TYPE ST185_Cylinders_e :
(
    Greifer_Patrone_Links,
    Greifer_Patrone_Rechts,
    Niederhalter_Deckel_Links,
    Niederhalter_Deckel_Rechts
);
END_TYPE

(* stored: Version 1.1.0.1, ProductVersion 3.1.4024.6
   EnumerationTextList ST185_Cylinders_e: Id {0a181d9d-b3e8-47b9-ba4f-bedc892e2da4} *)
